PROGRAM MAIN
VAR
END_VAR

PRG_HEARTBEAT();
PRG_PROTOTYPE();

END_PROGRAM

(* stored: Version 1.1.0.1, ProductVersion 3.1.4022.12
   POU MAIN: Id {21406078-f4f5-48e4-9241-b5d9a399051c}, SpecialFunc None *)
